// TIA Portal V17 export
// export: Created 2024-03-30T11:15:00.9360034Z, ExportSetting WithDefaults, DisplayName Totally Integrated Automation Portal, DisplayVersion V17, DisplayName TIA Portal Openness, DisplayVersion V17, DisplayName TIA Portal Version Control Interface, DisplayVersion V17, DisplayName STEP 7 Professional, DisplayVersion V17, DisplayName STEP 7 Safety, DisplayVersion V17, DisplayName WinCC Advanced, DisplayVersion V17
TYPE "typ_Config_Environment_Sensor"
// stored: IsFailsafeCompliant false
   STRUCT
      ldt_ts : LDT;
      di_period : DInt;
   END_STRUCT;
END_TYPE
